{attribute 'qualified_only'}
{attribute 'strict'}
TYPE ESequences :
(
	empty := 0,
	sample_sequence := 1
) UINT;
END_TYPE

(* stored: Version 1.1.0.1
   DUT ESequences: Id {810bdf63-30b5-4cb0-a38c-20ab681b03ec} *)
